{attribute 'GeneratedUsingTerminal: EL5042-0000-0016'}
{attribute addProperty BoxType "EL5042-0000-0016"}
{attribute addProperty Id "FB_Inputs_Channel_1AT %I*FB_Inputs_Channel_7405098814FB_Inputs_Channel_2AT %I*FB_Inputs_Channel_7405098814WcStateAT %I*WcState_9091E0EB2InfoDataAT %I*InfoData_94A18F5E2"}
{attribute addProperty CRC "450401401"}
{attribute addProperty Size "32"}
TYPE EL5042_1AD89479 EXTENDS EtcSlaveTerminalBase_947E5A46 :
STRUCT
	{attribute addProperty Name "FB_Inputs_Channel_1"}
	FB_Inputs_Channel_1 : FB_Inputs_Channel_74050988;
	{attribute addProperty Name "FB_Inputs_Channel_2"}
	FB_Inputs_Channel_2 : FB_Inputs_Channel_74050988;
	{attribute addProperty Name "WcState"}
	WcState : WcState_9091E0EB;
	{attribute addProperty Name "InfoData"}
	InfoData : InfoData_94A18F5E;
END_STRUCT
END_TYPE

(* stored: Version 1.2.0.0, ProductVersion 3.1.4024.9
   DUT EL5042_1AD89479: Id {096c747c-3cd4-4423-b707-9e26972f6f1f} *)
